// TIA Portal V21 export
DATA_BLOCK "PhtTimer"   // DB1216
{ S7_Optimized_Access := 'FALSE' }
// stored: AutoNumber false
   VAR
      "ReportData ResetTImer" : IEC_TIMER;
      "TIMER" { S7_SetPoint := 'True'} : IEC_TIMER;
      HVEventsTimer : Array[0..20] of IEC_TIMER;
      PhtTime1 { S7_SetPoint := 'True'} : IEC_TIMER;
      PhtTime2 { S7_SetPoint := 'True'} : IEC_TIMER;
      PhtTime3 { S7_SetPoint := 'True'} : IEC_TIMER;
      PhtTime4 { S7_SetPoint := 'True'} : IEC_TIMER;
      PhtTime5 { S7_SetPoint := 'True'} : IEC_TIMER;
      PhtTime6 { S7_SetPoint := 'True'} : IEC_TIMER;
      PhtTime7 { S7_SetPoint := 'True'} : IEC_TIMER;
      PhtTime8 { S7_SetPoint := 'True'} : IEC_TIMER;
      PhtTime9 { S7_SetPoint := 'True'} : IEC_TIMER;
      PhtTime10 { S7_SetPoint := 'True'} : IEC_TIMER;
   END_VAR
BEGIN
END_DATA_BLOCK
